FUNCTION_BLOCK DO_ACTION (* Basic Function Block Type *)
  (* Standard: 61499-2 *)
  (* Version 0.0, 2/8/2023, brink, Flexbridge AB, Template *)
  PACKAGE UAO.Hackathon;
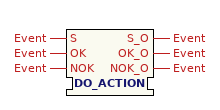
  EVENT_INPUT
    S; (* Action start *)
    OK; (* Action done *)
    NOK;
  END_EVENT
  EVENT_OUTPUT
    S_O;
    OK_O;
    NOK_O;
  END_EVENT
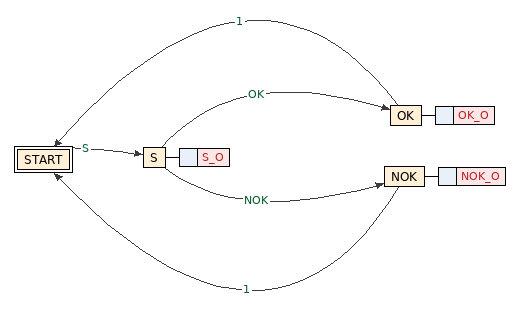
  EC_STATES
    START; (* Initial State *)
    S : -> S_O;
    OK : -> OK_O;
    NOK : -> NOK_O;
  END_STATES
  EC_TRANSITIONS
    START TO S := S;
    S TO OK := OK;
    OK TO START := 1;
    S TO NOK := NOK;
    NOK TO START := 1;
  END_TRANSITIONS
  ALGORITHM INIT IN ST:
;
  END_ALGORITHM
END_FUNCTION_BLOCK
